PROGRAM MAIN
VAR
	
// Inputs
	HoofdSchakelaar: BOOL;
	prevDrukKnop: BOOL;
	DrukKnop: BOOL;
	Teller: INT;

// Outputs
	MotorLinks: BOOL;
	MotorRechts: BOOL;

END_VAR

(*
Motor starten met één drukknop (4 regels code)

Schrijf een programma om een motor [ Relais voor MotorLinks en MotorRechts ] te starten en te stoppen met één drukknop. 
De installatie zal pas werken als een hoofdschakelaar AAN staat.

    1e druk op de drukknop:	start links draaiend
    2e druk op de drukknop:	stop
    3e druk op de drukknop:	start rechts draaiend
    4e druk op de drukknop:	stop
*)

IF HoofdSchakelaar AND NOT prevDrukKnop AND DrukKnop THEN Teller := (Teller + 1) MOD 4; END_IF;
prevDrukKnop := DrukKnop;
MotorLinks := HoofdSchakelaar AND Teller = 1;
MotorRechts := HoofdSchakelaar AND Teller = 3;

END_PROGRAM

(* stored: Version 1.1.0.1, ProductVersion 3.1.4024.12
   POU MAIN: Id {07ce2104-48e2-40da-9fdc-74ccafe19003}, SpecialFunc None *)
